Yaskawa INFORM job: TCP-R2-KM.JBI

/JOB
//NAME TCP-R2-KM
//POS
///NPOS 24,24,24,0,0,0
///TOOL 0
///POSTYPE PULSE
///PULSE
C00000=2000,-113621,-91818,-15,89172,2
C00001=1802,-98140,-117790,-24,33313,-69
C00002=34779,-39620,-121121,-28408,61723,-65986
C00003=45042,-191,-94167,-35731,66971,-65190
C00004=53299,13632,-81534,-51542,71819,-62128
C00005=52848,13301,-80689,-51384,71243,-61923
C00006=50539,10219,-83501,-49663,70653,-62263
C00007=55746,10958,-91670,-52283,75572,-63670
C00008=-11677,53872,-41789,75964,93315,-41146
C00009=-9980,52451,-42655,74912,92564,-41135
C00010=-10335,56513,-47190,75579,94081,-38976
C00011=-10335,56513,-47190,75579,94081,-38976
C00012=2000,-113621,-91818,-15,89172,2
C00013=11976,-46655,-12184,-57649,108255,24508
C00014=-3969,-3525,20856,-63185,99566,20978
C00015=-5656,12281,51754,-73749,98051,26640
C00016=-6188,12651,52672,-73883,97607,26759
C00017=-6205,11749,51475,-73933,97682,26634
C00018=-6188,11865,51256,-73960,97752,26549
C00019=-6168,12798,52434,-73910,97689,26660
C00020=-6188,12651,52672,-73883,97607,26759
C00021=-768,12236,51918,-71858,101051,27186
C00022=11976,-46655,-12184,-57649,108255,24508
C00023=2000,-113621,-91818,-15,89172,2
BC00000=87190,689488,413413
BC00001=203697,689488,1066499
BC00002=266323,689488,1066499
BC00003=266323,689488,1066499
BC00004=266323,689488,1066499
BC00005=266323,689488,1066499
BC00006=266323,689488,1066499
BC00007=266323,689488,1066499
BC00008=266323,689488,1066499
BC00009=266323,689488,1066499
BC00010=266323,689488,1066499
BC00011=104980,689488,1066499
BC00012=87190,689488,413413
BC00013=227836,769130,413410
BC00014=227836,769130,413410
BC00015=227836,769130,413410
BC00016=227836,769130,413410
BC00017=227836,769130,413410
BC00018=227836,769130,413410
BC00019=227836,769130,413410
BC00020=227836,769130,413410
BC00021=227836,769130,413410
BC00022=227836,769130,413410
BC00023=87190,689488,413413
EC00000=3,2
EC00001=3,2
EC00002=3,2
EC00003=3,2
EC00004=3,2
EC00005=3,2
EC00006=3,2
EC00007=3,2
EC00008=3,2
EC00009=3,2
EC00010=3,2
EC00011=3,2
EC00012=3,2
EC00013=3,2
EC00014=3,2
EC00015=3,2
EC00016=3,2
EC00017=3,2
EC00018=3,2
EC00019=3,2
EC00020=3,2
EC00021=3,2
EC00022=3,2
EC00023=3,2
//INST
///DATE 2024/03/19 19:22
///ATTR SC,RW
///GROUP1 RB1,BS1
///GROUP2 ST1
NOP
SFTOF3D
SSFTOF
SFTOF
MOVJ C00000 BC00000 VJ=100.00  +MOVJ EC00000 VJ=100.00
MOVJ C00001 BC00001 VJ=100.00  +MOVJ EC00001 VJ=100.00
MOVJ C00002 BC00002 VJ=100.00  +MOVJ EC00002 VJ=100.00
MOVJ C00003 BC00003 VJ=100.00  +MOVJ EC00003 VJ=100.00
MOVL C00004 BC00004 V=83.3  +MOVJ EC00004 VJ=100.00
'P1
MOVL C00005 BC00005 V=16.7 PL=0  +MOVJ EC00005 VJ=100.00
PAUSE
'P2
MOVL C00006 BC00006 V=16.7  +MOVJ EC00006 VJ=100.00
PAUSE
MOVL C00007 BC00007 V=83.3  +MOVJ EC00007 VJ=100.00
MOVL C00008 BC00008 V=83.3  +MOVJ EC00008 VJ=100.00
'P3
MOVL C00009 BC00009 V=16.7  +MOVJ EC00009 VJ=100.00
PAUSE
MOVL C00010 BC00010 V=250.0  +MOVJ EC00010 VJ=100.00
MOVJ C00011 BC00011 VJ=100.00  +MOVJ EC00011 VJ=100.00
MOVJ C00012 BC00012 VJ=100.00  +MOVJ EC00012 VJ=100.00
MOVJ C00013 BC00013 VJ=100.00  +MOVJ EC00013 VJ=100.00
MOVJ C00014 BC00014 VJ=100.00  +MOVJ EC00014 VJ=100.00
MOVJ C00015 BC00015 VJ=15.00  +MOVJ EC00015 VJ=100.00
PAUSE
MOVC C00016 BC00016 V=3.3  +MOVJ EC00016 VJ=15.00
MOVC C00017 BC00017 V=3.3  +MOVJ EC00017 VJ=15.00
MOVC C00018 BC00018 V=3.3  +MOVJ EC00018 VJ=15.00
MOVC C00019 BC00019 V=3.3  +MOVJ EC00019 VJ=15.00
MOVC C00020 BC00020 V=3.3  +MOVJ EC00020 VJ=15.00
MOVJ C00021 BC00021 VJ=15.00  +MOVJ EC00021 VJ=15.00
MOVJ C00022 BC00022 VJ=50.00  +MOVJ EC00022 VJ=15.00
MOVJ C00023 BC00023 VJ=100.00  +MOVJ EC00023 VJ=50.00
END
